(* CODESYS project tcl_UnitTestLibrary.library
   Company: Red Rock Controls Limited
   Description: AssertEquals_USINT added
   Version: 1.1.3.0
   Placeholder: tcl_UnitTestLibrary
   Author: Roger Christopher
   Title: tcl_UnitTestLibrary

Project tree, tasks and I/O mapping:
  libraries: Tc2_Standard, * (Beckhoff Automation GmbH); Tc2_System, * (Beckhoff Automation GmbH); Tc2_Utilities, * (Beckhoff Automation GmbH); Tc3_Module, * (Beckhoff Automation GmbH)
  Functions/
    function F_LogError [ST]
    function F_LogMessage [ST]
  String Utils/
    function FormatString1 [ST]
    function FormatString2 [ST]
    function FormatString3 [ST]
    function FormatStringEx1 [ST]
    function FormatStringEx2 [ST]
    function block StringSplitter [ST]: GetNext, GetRemainder, HasMore, Init
  Unit Test/
    function block T_UnitTestBase [ST]: AssertEquals_ANY, AssertEquals_BOOL, AssertEquals_BYTE, AssertEquals_DINT, AssertEquals_INT, AssertEquals_LINT, AssertEquals_LREAL, AssertEquals_PVOID, AssertEquals_REAL, AssertEquals_STRING, AssertEquals_UDINT, AssertEquals_UINT, AssertEquals_ULINT, AssertEquals_USINT, AssertIsFalse, AssertIsTrue, Fail, FB_init, Init, RunTest, Name, TestCompleted, TestFailed
  Version/
    global variables Global_Version
  global variables Globals
*)

// Version/Global_Version
{attribute 'TcGenerated'}
{attribute 'no-analysis'}
{attribute 'linkalways'}
// This function has been automatically generated from the project information.
VAR_GLOBAL CONSTANT
	{attribute 'const_non_replaced'}
	stLibVersion_tcl_UnitTestLibrary : ST_LibVersion := (iMajor := 1, iMinor := 1, iBuild := 3, iRevision := 0, nFlags := 0, sVersion := '1.1.3.0');
END_VAR

// Globals
{attribute 'qualified_only'}
VAR_GLOBAL

END_VAR

// Functions/F_LogError
FUNCTION INTERNAL F_LogError : BOOL
VAR_INPUT
    Source  : T_MaxString;
    Message : T_MaxString;
END_VAR
VAR
END_VAR

ADSLOGSTR(msgCtrlMask := ADSLOG_MSGTYPE_STRING OR ADSLOG_MSGTYPE_ERROR OR ADSLOG_MSGTYPE_LOG,
          msgFmtStr   := FormatStringEx2('%s : %s', Source, Message),
          strArg      := '');

END_FUNCTION

// String Utils/FormatStringEx2
{attribute 'hide'}
FUNCTION INTERNAL FormatStringEx2 : T_MaxString
VAR_INPUT
	Format	: T_MaxString;
	arg1	: T_MaxString;
	arg2	: T_MaxString;
END_VAR
VAR
    FB_FormatString1 : FB_FormatString;
END_VAR

FB_FormatString1(sFormat := Format,
                 arg1    := F_STRING(arg1),
                 arg2    := F_STRING(arg2),
                 arg3    :=,
                 arg4    :=,
                 arg5    :=,
                 arg6    :=,
                 arg7    :=,
                 arg8    :=,
                 arg9    :=,
                 arg10   :=,
                 bError  =>,
                 nErrId  =>,
                 sOut    => FormatStringEx2);

END_FUNCTION

// Functions/F_LogMessage
FUNCTION INTERNAL F_LogMessage : BOOL
VAR_INPUT
    Source  : T_MaxString;
    Message : T_MaxString;
END_VAR
VAR
END_VAR

ADSLOGSTR(msgCtrlMask := ADSLOG_MSGTYPE_STRING OR ADSLOG_MSGTYPE_HINT OR ADSLOG_MSGTYPE_LOG,
          msgFmtStr   := FormatStringEx2('%s : %s', Source, Message),
          strArg      := '');

END_FUNCTION

// String Utils/FormatString1
{attribute 'hide'}
FUNCTION INTERNAL FormatString1 : T_MaxString
VAR_INPUT
	Format	: T_MaxString;
	arg1	: T_Arg;
END_VAR
VAR
    FB_FormatString1 : FB_FormatString;
END_VAR

FB_FormatString1(sFormat := Format,
                 arg1    := arg1,
                 arg2    :=,
                 arg3    :=,
                 arg4    :=,
                 arg5    :=,
                 arg6    :=,
                 arg7    :=,
                 arg8    :=,
                 arg9    :=,
                 arg10   :=,
                 bError  =>,
                 nErrId  =>,
                 sOut    => FormatString1);

END_FUNCTION

// String Utils/FormatString2
{attribute 'hide'}
FUNCTION INTERNAL FormatString2 : T_MaxString
VAR_INPUT
	Format	: T_MaxString;
	arg1	: T_Arg;
	arg2	: T_Arg;
END_VAR
VAR
    FB_FormatString1 : FB_FormatString;
END_VAR

FB_FormatString1(sFormat := Format,
                 arg1    := arg1,
                 arg2    := arg2,
                 arg3    :=,
                 arg4    :=,
                 arg5    :=,
                 arg6    :=,
                 arg7    :=,
                 arg8    :=,
                 arg9    :=,
                 arg10   :=,
                 bError  =>,
                 nErrId  =>,
                 sOut    => FormatString2);

END_FUNCTION

// String Utils/FormatString3
{attribute 'hide'}
FUNCTION INTERNAL FormatString3 : T_MaxString
VAR_INPUT
	Format	: T_MaxString;
	arg1	: T_Arg;
	arg2	: T_Arg;
	arg3	: T_Arg;
END_VAR
VAR
    FB_FormatString1 : FB_FormatString;
END_VAR

FB_FormatString1(sFormat := Format,
                 arg1    := arg1,
                 arg2    := arg2,
                 arg3    := arg3,
                 arg4    :=,
                 arg5    :=,
                 arg6    :=,
                 arg7    :=,
                 arg8    :=,
                 arg9    :=,
                 arg10   :=,
                 bError  =>,
                 nErrId  =>,
                 sOut    => FormatString3);

END_FUNCTION

// String Utils/FormatStringEx1
{attribute 'hide'}
FUNCTION INTERNAL FormatStringEx1 : T_MaxString
VAR_INPUT
	Format	: T_MaxString;
	arg1	: T_MaxString;
END_VAR
VAR
    FB_FormatString1 : FB_FormatString;
END_VAR


FB_FormatString1(sFormat := Format,
                 arg1    := F_STRING(arg1),
                 arg2    :=,
                 arg3    :=,
                 arg4    :=,
                 arg5    :=,
                 arg6    :=,
                 arg7    :=,
                 arg8    :=,
                 arg9    :=,
                 arg10   :=,
                 bError  =>,
                 nErrId  =>,
                 sOut    => FormatStringEx1);

END_FUNCTION

// String Utils/StringSplitter
{attribute 'hide'}
FUNCTION_BLOCK INTERNAL StringSplitter
VAR
	SubjectString : TC2_SYSTEM.T_MaxString;
	Delimiter : STRING;
	Delimiter1 : STRING;
	Delimiter2 : STRING;
	NextDelimiterPosition : INT;
	NextDelimiter1Position : INT;
	NextDelimiter2Position : INT;
END_VAR

METHOD GetNext : STRING(255)
VAR_INPUT
END_VAR
VAR
	RemainingLength: INT;
END_VAR
NextDelimiter1Position := FIND(SubjectString , Delimiter1);
NextDelimiter2Position := FIND(SubjectString , Delimiter2);

IF NextDelimiter1Position = 0 THEN
    // use Delimiter 2 position , even if zero...
    NextDelimiterPosition := NextDelimiter2Position;
    Delimiter := Delimiter2;
    
ELSIF NextDelimiter2Position = 0 THEN
    // use Delimiter 1 position , non-zero...
    NextDelimiterPosition := NextDelimiter1Position;
    Delimiter := Delimiter1;

ELSE
    // Both delimters found - use the one nearest the start of the string...
    IF NextDelimiter1Position < NextDelimiter2Position THEN
        NextDelimiterPosition := NextDelimiter1Position;
        Delimiter := Delimiter1;
    ELSE
        NextDelimiterPosition := NextDelimiter2Position;
        Delimiter := Delimiter2;
	END_IF
END_IF

IF NextDelimiterPosition > 0 THEN // delimitter found
    
    // extract next sub-string
	GetNext := LEFT(SubjectString,NextDelimiterPosition - 1);
    
    // remove sub-string from subject string
	RemainingLength := LEN(SubjectString) - NextDelimiterPosition - LEN(Delimiter) + 1;
	SubjectString := RIGHT(SubjectString,RemainingLength);
    
//    // strip any delimitters from front of remaining string
//    WHILE FIND(SubjectString,Delimiter1) = 1 DO
//        SubjectString := RIGHT(SubjectString,LEN(SubjectString) - LEN(Delimiter1));
//	END_WHILE
//    WHILE FIND(SubjectString,Delimiter2) = 1 DO
//        SubjectString := RIGHT(SubjectString,LEN(SubjectString) - LEN(Delimiter2));
//	END_WHILE
ELSE
	GetNext := SubjectString; // return what is left
	SubjectString := '';
END_IF
END_METHOD

METHOD GetRemainder : STRING(255)
GetRemainder := SubjectString; // return what is left
SubjectString := '';
END_METHOD

METHOD HasMore : BOOL
VAR_INPUT
END_VAR
HasMore := SubjectString <> '';
END_METHOD

METHOD Init
VAR_INPUT
		Str : TC2_SYSTEM.T_MaxString;
		Delim1 : STRING;
		Delim2 : STRING;
END_VAR
SubjectString := Str;
NextDelimiterPosition := 0;
Delimiter1 := Delim1;
Delimiter2 := Delim2;
END_METHOD

END_FUNCTION_BLOCK

// Unit Test/T_UnitTestBase
{attribute 'reflection'}
FUNCTION_BLOCK ABSTRACT T_UnitTestBase
VAR
    {attribute 'instance-path'}
    {attribute 'no_init'}
    {attribute 'analysis' := '-33'} // Inhibit unused variable warning
    InstanceName : T_MaxString;     // Initialised with the instance name

    Project  : T_MaxString;
    Plc      : T_MaxString;
    TestName : T_MaxString;

    _TestCompleted : BOOL;
    _TestFailed    : BOOL;
    State          : INT;
    CycleCount     : UDINT;
    Retest         : BOOL;
END_VAR

METHOD PROTECTED AssertEquals_ANY : BOOL
VAR_INPUT
    Expected : ANY;
    Actual   : ANY;
    Message  : T_MaxString;
END_VAR
VAR
    ComparisonResult : DINT;
END_VAR
ComparisonResult := MEMCMP(pBuf1 := Expected.pValue,
                           pBuf2 := Actual.pValue,
                           n     := DINT_TO_UDINT(Actual.diSize));

IF Expected.TypeClass <> Actual.TypeClass THEN
    F_LogError(TestName, FormatStringEx1('Assertion Failed - %s', Message));
    TestFailed    := TRUE;
    TestCompleted := TRUE;
    RETURN;

ELSIF Expected.diSize <> Actual.diSize THEN
    F_LogError(TestName, FormatStringEx1('Assertion Failed - %s', Message));
    TestFailed    := TRUE;
    TestCompleted := TRUE;
    RETURN;

ELSIF ComparisonResult <> 0 THEN
    F_LogError(TestName, FormatStringEx1('Assertion Failed - %s', Message));
    TestFailed    := TRUE;
    TestCompleted := TRUE;
    RETURN;
END_IF

AssertEquals_ANY := TRUE;
END_METHOD

METHOD PROTECTED AssertEquals_BOOL : BOOL
VAR_INPUT
    Expected : BOOL;
    Actual   : BOOL;
    Message  : T_MaxString;
END_VAR
VAR
    ExpectedAsString : STRING;
    ActualAsString   : STRING;
END_VAR
IF Expected <> Actual THEN
	ExpectedAsString := BOOL_TO_STRING(Expected);
	ActualAsString := BOOL_TO_STRING(Actual);
    F_LogError(TestName,
               FormatString3('%s: expected=%s, actual=%s',
                             F_STRING(Message),
                             F_STRINGEX(ExpectedAsString),
                             F_STRINGEX(ActualAsString)));
    TestFailed    := TRUE;
    TestCompleted := TRUE;
    RETURN;
END_IF

AssertEquals_BOOL := TRUE;
END_METHOD

METHOD PROTECTED AssertEquals_BYTE : BOOL
VAR_INPUT
    Expected : BYTE;
    Actual   : BYTE;
    Message  : T_MaxString;
END_VAR
IF Expected <> Actual THEN
    F_LogError(TestName,
               FormatString3('%s: expected=0x%.2X, actual=0x%.2X',
                             F_STRING(Message),
                             F_BYTE(Expected),
                             F_BYTE(Actual)));
    TestFailed    := TRUE;
    TestCompleted := TRUE;
    RETURN;
END_IF

AssertEquals_BYTE := TRUE;
END_METHOD

METHOD PROTECTED AssertEquals_DINT : BOOL
VAR_INPUT
    Expected : DINT;
    Actual   : DINT;
    Message  : T_MaxString;
END_VAR
IF Expected <> Actual THEN
    F_LogError(TestName,
               FormatString3('%s: expected=%d, actual=%d',
                             F_STRING(Message),
                             F_DINT(Expected),
                             F_DINT(Actual)));
    TestFailed    := TRUE;
    TestCompleted := TRUE;
    RETURN;
END_IF

AssertEquals_DINT := TRUE;
END_METHOD

METHOD PROTECTED AssertEquals_INT : BOOL
VAR_INPUT
    Expected : INT;
    Actual   : INT;
    Message  : T_MaxString;
END_VAR
IF Expected <> Actual THEN
    F_LogError(TestName,
               FormatString3('%s: expected=%d, actual=%d',
                             F_STRING(Message),
                             F_INT(Expected),
                             F_INT(Actual)));
    TestFailed    := TRUE;
    TestCompleted := TRUE;
    RETURN;
END_IF

AssertEquals_INT := TRUE;
END_METHOD

METHOD PROTECTED AssertEquals_LINT : BOOL
VAR_INPUT
    Expected : LINT;
    Actual   : LINT;
    Message  : T_MaxString;
END_VAR
IF Expected <> Actual THEN
    F_LogError(TestName,
               FormatString3('%s: expected=%d, actual=%d',
                             F_STRING(Message),
                             F_LINT(Expected),
                             F_LINT(Actual)));
    TestFailed    := TRUE;
    TestCompleted := TRUE;
    RETURN;
END_IF

AssertEquals_LINT := TRUE;
END_METHOD

METHOD PROTECTED AssertEquals_LREAL : BOOL
VAR_INPUT
    Expected : LREAL;
    Actual   : LREAL;
    Delta    : LREAL;
    Message  : T_MaxString;
END_VAR
IF ABS(Expected - Actual) > Delta THEN
    F_LogError(TestName,
               FormatString3('%s: expected= %.3f, actual= %.3f',
                             F_STRING(Message),
                             F_LREAL(Expected),
                             F_LREAL(Actual)));
    TestFailed    := TRUE;
    TestCompleted := TRUE;
    RETURN;
END_IF

AssertEquals_LREAL := TRUE;
END_METHOD

METHOD PROTECTED AssertEquals_PVOID : BOOL
VAR_INPUT
    Expected : PVOID;
    Actual   : PVOID;
    Message  : T_MaxString;
END_VAR
IF Expected <> Actual THEN
    F_LogError(TestName,
               FormatString3('%s: expected=%d, actual=%d',
                             F_STRING(Message),
                             F_PVOID(Expected),
                             F_PVOID(Actual)));
    TestFailed    := TRUE;
    TestCompleted := TRUE;
    RETURN;
END_IF

AssertEquals_PVOID := TRUE;
END_METHOD

METHOD PROTECTED AssertEquals_REAL : BOOL
VAR_INPUT
    Expected : REAL;
    Actual   : REAL;
    Delta    : REAL;
    Message  : T_MaxString;
END_VAR
IF ABS(Expected - Actual) > Delta THEN
    F_LogError(TestName,
               FormatString3('%s: expected=%.3f, actual=%.3f',
                             F_STRING(Message),
                             F_REAL(Expected),
                             F_REAL(Actual)));
    TestFailed    := TRUE;
    TestCompleted := TRUE;
    RETURN;
END_IF

AssertEquals_REAL := TRUE;
END_METHOD

METHOD PROTECTED AssertEquals_STRING : BOOL
VAR_INPUT
    Expected : T_MaxString;
    Actual   : T_MaxString;
    Message  : T_MaxString;
END_VAR
IF Expected <> Actual THEN
    F_LogError(TestName,
               FormatString3('%s: expected=%s, actual=%s',
                             F_STRING(Message),
                             F_STRING(Expected),
                             F_STRING(Actual)));
    TestFailed    := TRUE;
    TestCompleted := TRUE;
    RETURN;
END_IF

AssertEquals_STRING := TRUE;
END_METHOD

METHOD PROTECTED AssertEquals_UDINT : BOOL
VAR_INPUT
    Expected : UDINT;
    Actual   : UDINT;
    Message  : T_MaxString;
END_VAR
IF Expected <> Actual THEN
    F_LogError(TestName,
               FormatString3('%s: expected=%d, actual=%d',
                             F_STRING(Message),
                             F_UDINT(Expected),
                             F_UDINT(Actual)));
    TestFailed    := TRUE;
    TestCompleted := TRUE;
    RETURN;
END_IF

AssertEquals_UDINT := TRUE;
END_METHOD

METHOD PROTECTED AssertEquals_UINT : BOOL
VAR_INPUT
    Expected : UINT;
    Actual   : UINT;
    Message  : T_MaxString;
END_VAR
IF Expected <> Actual THEN
    F_LogError(TestName,
               FormatString3('%s: expected=%d, actual=%d',
                             F_STRING(Message),
                             F_UINT(Expected),
                             F_UINT(Actual)));
    TestFailed    := TRUE;
    TestCompleted := TRUE;
    RETURN;
END_IF

AssertEquals_UINT := TRUE;
END_METHOD

METHOD PROTECTED AssertEquals_ULINT : BOOL
VAR_INPUT
    Expected : ULINT;
    Actual   : ULINT;
    Message  : T_MaxString;
END_VAR
IF Expected <> Actual THEN
    F_LogError(TestName,
               FormatString3('%s: expected=%d, actual=%d',
                             F_STRING(Message),
                             F_ULINT(Expected),
                             F_ULINT(Actual)));
    TestFailed    := TRUE;
    TestCompleted := TRUE;
    RETURN;
END_IF

AssertEquals_ULINT := TRUE;
END_METHOD

METHOD PROTECTED AssertEquals_USINT : BOOL
VAR_INPUT
    Expected : USINT;
    Actual   : USINT;
    Message  : T_MaxString;
END_VAR
IF Expected <> Actual THEN
    F_LogError(TestName,
               FormatString3('%s: expected=%d, actual=%d',
                             F_STRING(Message),
                             F_USINT(Expected),
                             F_USINT(Actual)));
    TestFailed    := TRUE;
    TestCompleted := TRUE;
    RETURN;
END_IF

AssertEquals_USINT := TRUE;
END_METHOD

METHOD PROTECTED AssertIsFalse : BOOL
VAR_INPUT
    Condition : BOOL;
    Message   : T_MaxString;
END_VAR
IF Condition THEN
    F_LogError(TestName,
               FormatString1('%s: expected=FALSE, actual=TRUE',
                             F_STRING(Message)));
    TestFailed    := TRUE;
    TestCompleted := TRUE;
    RETURN;
END_IF

AssertIsFalse := TRUE;
END_METHOD

METHOD PROTECTED AssertIsTrue : BOOL
VAR_INPUT
    Condition : BOOL;
    Message   : T_MaxString;
END_VAR
IF NOT Condition THEN
    F_LogError(TestName,
               FormatString1('%s: expected=TRUE, actual=FALSE',
                             F_STRING(Message)));
    TestFailed    := TRUE;
    TestCompleted := TRUE;
    RETURN;
END_IF

AssertIsTrue := TRUE;
END_METHOD

METHOD Fail
VAR_INPUT
    Message : T_MaxString;
END_VAR
F_LogError(TestName, FormatStringEx1('Test Failed - %s', Message));
TestFailed    := TRUE;
TestCompleted := TRUE;
END_METHOD

METHOD FB_init : BOOL
VAR_INPUT
	bInitRetains : BOOL; // if TRUE, the retain variables are initialized (warm start / cold start)
	bInCopyCode : BOOL;  // if TRUE, the instance afterwards gets moved into the copy code (online change)
END_VAR
THIS^.Init();
END_METHOD

{attribute 'call_after_online_change_slot' := '1000'}
METHOD Init
VAR
    StringSplitter : StringSplitter;
END_VAR
StringSplitter.Init(Str    := InstanceName,
                    Delim1 := '.',
                    Delim2 := '');

IF StringSplitter.HasMore() THEN
    Project := StringSplitter.GetNext();
    Plc     := StringSplitter.GetNext();
END_IF

WHILE StringSplitter.HasMore() DO
    TestName := StringSplitter.GetNext(); // gets last chunk, which is Test Name
END_WHILE

State          := 0;
CycleCount     := 0;
_TestFailed    := FALSE;
_TestCompleted := FALSE;
Retest         := FALSE;
END_METHOD

{attribute 'analysis' := '-33'} // inhibit unused variable warning
METHOD ABSTRACT RunTest
END_METHOD

PROPERTY Name : T_MaxString
GET
Name := TestName;
END_GET
END_PROPERTY

PROPERTY TestCompleted : BOOL
GET
PUBLIC
TestCompleted := _TestCompleted;
END_GET
SET
PROTECTED
_TestCompleted := TestCompleted;
END_SET
END_PROPERTY

PROPERTY TestFailed : BOOL
GET
PUBLIC
TestFailed := _TestFailed;
END_GET
SET
PROTECTED
_TestFailed := TestFailed;
END_SET
END_PROPERTY

END_FUNCTION_BLOCK
